{attribute addProperty BoxType "EK1100-0000-0018"}
{attribute addProperty Id "Beckhoff_EK15xxEK1122Beckhoff_EK15xxEK1122_8310362454468A_0025_EK1561_0000_0018EK1561_179A0949162A_0024_EK1561_0000_0017EK1561_179A0949162A_0023_EK1561_0000_0016EK1561_179A0949162A_0019_EK1521_0010_0020EK1521_179A0949162A_0018_EK1521_0010_0019EK1521_179A0949162A_0017_EK1521_0010_0018EK1521_179A0949162A_0016_EK1521_0010_0017EK1521_179A0949162A_0015_EK1521_0010_0016EK1521_179A0949162A_0014_EK1521_0000_0021EK1521_179A0949162A_0013_EK1521_0000_0020EK1521_179A0949162A_0012_EK1521_0000_0019EK1521_179A0949162A_0011_EK1521_0000_0018EK1521_179A0949162A_0010_EK1521_0000_0017EK1521_179A0949162A_0009_EK1521_0000_0016EK1521_179A0949162"}
{attribute addProperty CRC "3734597087"}
{attribute addProperty SizeInBites "768"}
{attribute addProperty SizeInBytes "96"}
TYPE Beckhoff_EK15xx_DE996DDF EXTENDS EK1100_179A0949 :
STRUCT
	{attribute addProperty Name "Beckhoff_EK15xxEK1122"}
	Beckhoff_EK15xxEK1122 : Beckhoff_EK15xxEK1122_83103624;
	{attribute addProperty Name "A_0025_EK1561_0000_0018"}
	A_0025_EK1561_0000_0018 : EK1561_179A0949;
	{attribute addProperty Name "A_0024_EK1561_0000_0017"}
	A_0024_EK1561_0000_0017 : EK1561_179A0949;
	{attribute addProperty Name "A_0023_EK1561_0000_0016"}
	A_0023_EK1561_0000_0016 : EK1561_179A0949;
	{attribute addProperty Name "A_0019_EK1521_0010_0020"}
	A_0019_EK1521_0010_0020 : EK1521_179A0949;
	{attribute addProperty Name "A_0018_EK1521_0010_0019"}
	A_0018_EK1521_0010_0019 : EK1521_179A0949;
	{attribute addProperty Name "A_0017_EK1521_0010_0018"}
	A_0017_EK1521_0010_0018 : EK1521_179A0949;
	{attribute addProperty Name "A_0016_EK1521_0010_0017"}
	A_0016_EK1521_0010_0017 : EK1521_179A0949;
	{attribute addProperty Name "A_0015_EK1521_0010_0016"}
	A_0015_EK1521_0010_0016 : EK1521_179A0949;
	{attribute addProperty Name "A_0014_EK1521_0000_0021"}
	A_0014_EK1521_0000_0021 : EK1521_179A0949;
	{attribute addProperty Name "A_0013_EK1521_0000_0020"}
	A_0013_EK1521_0000_0020 : EK1521_179A0949;
	{attribute addProperty Name "A_0012_EK1521_0000_0019"}
	A_0012_EK1521_0000_0019 : EK1521_179A0949;
	{attribute addProperty Name "A_0011_EK1521_0000_0018"}
	A_0011_EK1521_0000_0018 : EK1521_179A0949;
	{attribute addProperty Name "A_0010_EK1521_0000_0017"}
	A_0010_EK1521_0000_0017 : EK1521_179A0949;
	{attribute addProperty Name "A_0009_EK1521_0000_0016"}
	A_0009_EK1521_0000_0016 : EK1521_179A0949;
END_STRUCT
END_TYPE

(* stored: Version 1.2.0.0, ProductVersion 3.1.4024.9
   DUT Beckhoff_EK15xx_DE996DDF: Id {a5349c98-50a8-4cd3-962a-5539d26a3659} *)
